PROGRAM prgComEffIO
VAR
	fbCom		: FB_MqttCommunicator_V4;
END_VAR

fbCom(
	bConnect				:= TRUE,
	strAuthKey				:=  'BMS99299754422' , 
	sUserName				:= '55916711-aa04-4806-95f6-e4f6430fad74', 
	sUserPassword			:= '029e75fe-43a2-4560-bcb6-707aba386d0a', 
	eSavePositionCertificate:= eSavePositionOnPLC.ePostionHardDisk, 
	time_HeartBeat_sec := T#15S,
	bConnected=> , 
	bError=> , 
	hrErrorCode=> , 
	eConnectionState=> , 
	eErrorMessage_Out=> );

END_PROGRAM

(* stored: Version 1.1.0.1, ProductVersion 3.1.4024.12
   POU prgComEffIO: Id {cbcd318b-bf51-484c-bcaa-d6efcdf43fe3}, SpecialFunc None *)
